FUNCTION TFPalletizerIsFormingAssigned : BOOL(*Funzione che restituisce valore VERO se non ci sono piazzole presenti con codice di formatura il codice di lavorazione indicati come Input*)
VAR_INPUT
	WorkArea : POINTER TO ARRAY [1..MAXAREA] OF TFMachinePalletizer_WorkArea;
	WorkAreaState : POINTER TO ARRAY [1..MAXAREA] OF TFMachinePalletizer_WorkAreaState;
	FCode : INT;
	PCode : INT;
END_VAR
VAR
	wa : INT;
	n : INT;
END_VAR
(*Funzione che restituisce valore VERO se non ci sono piazzole presenti con codice di formatura il codice di lavorazione indicati come Input*)

(*Funzione che restituisce valore VERO se non ci sono piazzole presenti con codice di formatura il codice di lavorazione indicati come Input*)
TFPalletizerIsFormingAssigned := FALSE; 

FOR wa:=1 TO MAXAREA DO
	IF WorkArea^[wa].Enable = 1 THEN
		(* Verifico se il codice è già stato assegnato *)
		IF WorkAreaState^[wa].F = FCode THEN
			IF WorkArea^[wa].Code = PCode OR WorkArea^[wa].Code = 0 THEN
				(* Verifico se la piazzola è in lavorazione *)
				(* Se è in lavorazione allora è inutile assegnarne un'altra con lo stesso codice *)
				IF WorkAreaState^[wa].State < WORKAREA_STATE_OCCUPIED_WORKED AND 
					WorkAreaState^[wa].State > WORKAREA_STATE_FREE_DISABLED THEN
					TFPalletizerIsFormingAssigned := TRUE;
					RETURN;
				END_IF
			END_IF
		END_IF
	END_IF
END_FOR

END_FUNCTION

(* stored: Version 1.1.0.1, ProductVersion 3.1.4024.11
   POU TFPalletizerIsFormingAssigned: Id {eec1639c-d5da-437a-93ab-cb23a694558d}, SpecialFunc None *)
